(* CODESYS project cylinders_initial.project

Project tree, tasks and I/O mapping:
  Device : CODESYS Control Win V3, 3S - Smart Software Solutions GmbH, version 3.5.16.0
    application Application
      libraries: Standard, * (System); CmpBitmapPool, * (System); Util, * (System)
      task MainTask (cyclic, interval 5 ms, priority 1) calls cylinder_ctrl_SFC
      task simulation (cyclic, interval t#20ms, priority 1) calls sim_logic
      task VISU_TASK (cyclic, interval 10 ms, priority 31) calls VisuElems.Visu_Prg
      visualisation Cylinders
      global variables IO
      control/
        program cylinder_ctrl [LD]
        function block CylinderFB [LD]
        function block LampCTRL [SFC]
        program cylinder_ctrl_SFC [LD]
        function block Sequence [SFC]
      simulation/
        program sim_logic [LD]
        function block cylSimulation [ST]
      image pool ImagePool
  libraries: VisuSymbols, 3.5.10.0 (System)
  5ce3da45-db07-42e7-a21c-a00fff4ed8f6|C:\Users\ryytt\OneDrive\Skrivbord\examensarbete\bakgrund.png
  5ce3da45-db07-42e7-a21c-a00fff4ed8f6|C:\Users\ryytt\OneDrive\Skrivbord\examensarbete\bakgrundv2.png
  text list GlobalTextList
*)

// Device/Application/IO
VAR_GLOBAL
	ixStart: BOOL; // the start switch and the button
 	ixStop: BOOL;  // the stop switch and the button
	ixReset: BOOL; // the reset switch
	ixB1: BOOL; // button B1
	ixB2: BOOL; // button B2
	ixIN10: BOOL; // the IN10 switch
	ixIN11: BOOL; // the IN11 switch
	ixCylinder1In: BOOL; // a sensor if cylinder 1 is in
	ixCylinder1Out: BOOL; // a sensor if cylinder 1 is in
	ixCylinder2In: BOOL; // a sensor if cylinder 1 is in
	ixCylinder2Out: BOOL; // a sensor if cylinder 1 is in
	ixCylinder3In: BOOL; // a sensor if cylinder 1 is in
	ixCylinder3Out: BOOL; // a sensor if cylinder 1 is in	
	ixEmergencyStop: BOOL := TRUE; // the emergency stop. If false, it is active

	qxLamp1: BOOL; // to control L1
	qxLamp2: BOOL; // to control L2
	qxLamp3: BOOL; // to ontorl L3
	qxLamp4: BOOL; // to control L4
	qxCylinder1: BOOL; // to extend cylinder 1
	qxCylinder2: BOOL; // to extend cylinder 2
	qxCylinder3: BOOL; // to extend cylinder 3
	ixCylinderIn_cyl23: BOOL;
	ixCylinderOut_cyl23: BOOL;
END_VAR

// Device/Application/control/cylinder_ctrl_SFC
PROGRAM cylinder_ctrl_SFC
VAR
	cylinder1: CylinderFB;
	cylinder2: CylinderFB;
	cylinder3: CylinderFB;
	
	sequence_ctrl1: Sequence;
	sequence_ctrl23: Sequence;
	
	LampCTRL_0: LampCTRL;
	lamp_testing: LampCTRL;
END_VAR

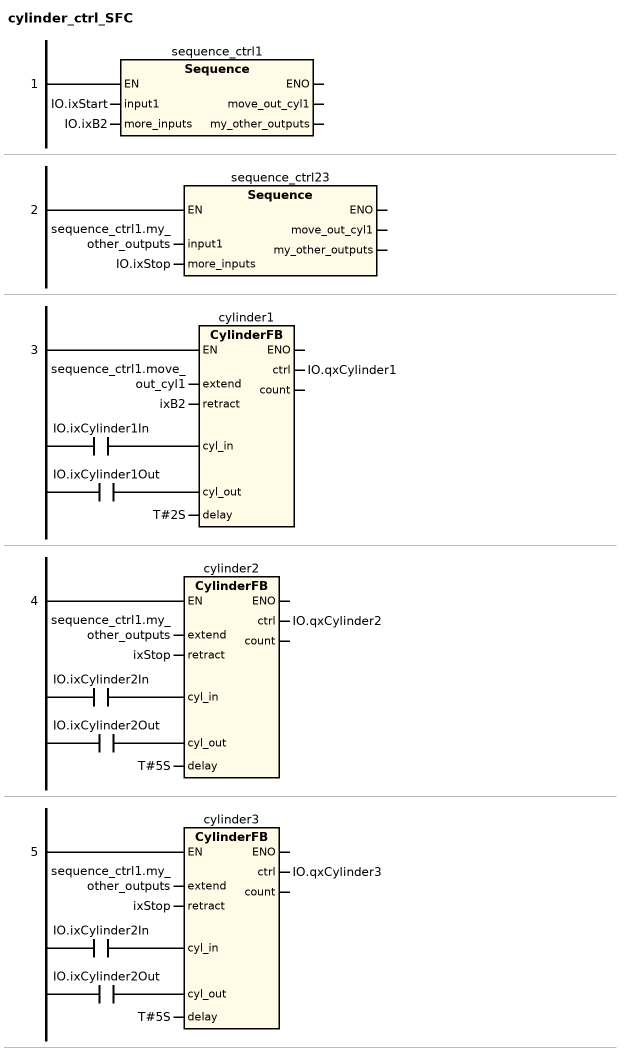
// NETWORK 1
sequence_ctrl1(input1 := IO.ixStart, more_inputs := IO.ixB2); // Sequence

// NETWORK 2
sequence_ctrl23(input1 := sequence_ctrl1.my_other_outputs, more_inputs := IO.ixStop); // Sequence

// NETWORK 3
cylinder1(
    extend := sequence_ctrl1.move_out_cyl1,
    retract := ixB2,
    cyl_in := IO.ixCylinder1In,
    cyl_out := IO.ixCylinder1Out,
    delay := T#2S,
    ctrl => IO.qxCylinder1); // CylinderFB

// NETWORK 4
cylinder2(
    extend := sequence_ctrl1.my_other_outputs,
    retract := ixStop,
    cyl_in := IO.ixCylinder2In,
    cyl_out := IO.ixCylinder2Out,
    delay := T#5S,
    ctrl => IO.qxCylinder2); // CylinderFB

// NETWORK 5
cylinder3(
    extend := sequence_ctrl1.my_other_outputs,
    retract := ixStop,
    cyl_in := IO.ixCylinder2In,
    cyl_out := IO.ixCylinder2Out,
    delay := T#5S,
    ctrl => IO.qxCylinder3); // CylinderFB

END_PROGRAM

// Device/Application/control/Sequence
FUNCTION_BLOCK Sequence
VAR_INPUT
	input1: BOOL;
	more_inputs: BOOL;
END_VAR
VAR_OUTPUT
	move_out_cyl1: BOOL;
	my_other_outputs: BOOL;
END_VAR
VAR
	init: BOOL := TRUE;
END_VAR

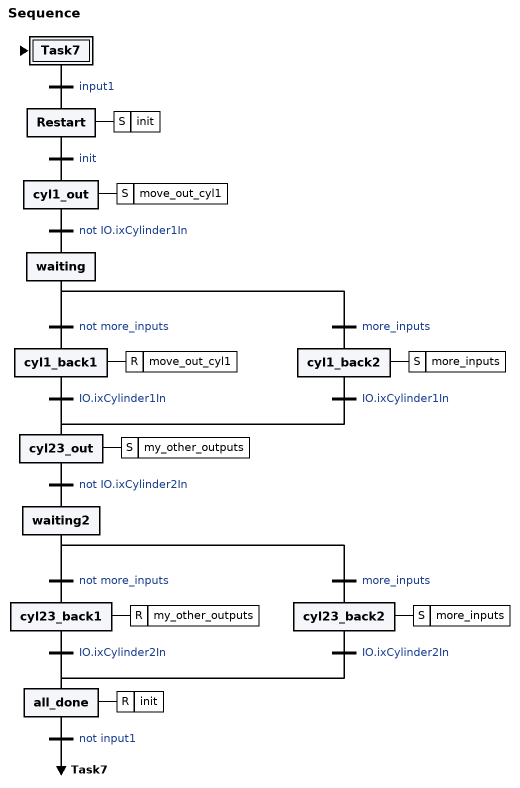
INITIAL_STEP Task7:
END_STEP
TRANSITION FROM Task7 TO Restart
    := input1;
END_TRANSITION
STEP Restart:
    init(S);
END_STEP
TRANSITION FROM Restart TO cyl1_out
    := init;
END_TRANSITION
STEP cyl1_out:
    move_out_cyl1(S);
END_STEP
TRANSITION FROM cyl1_out TO waiting
    := not IO.ixCylinder1In;
END_TRANSITION
STEP waiting:
END_STEP
TRANSITION FROM waiting TO cyl1_back1
    := not more_inputs;
END_TRANSITION
STEP cyl1_back1:
    move_out_cyl1(R);
END_STEP
TRANSITION FROM cyl1_back1 TO cyl23_out
    := IO.ixCylinder1In;
END_TRANSITION
TRANSITION FROM waiting TO cyl1_back2
    := more_inputs;
END_TRANSITION
STEP cyl1_back2:
    more_inputs(S);
END_STEP
TRANSITION FROM cyl1_back2 TO cyl23_out
    := IO.ixCylinder1In;
END_TRANSITION
STEP cyl23_out:
    my_other_outputs(S);
END_STEP
TRANSITION FROM cyl23_out TO waiting2
    := not IO.ixCylinder2In;
END_TRANSITION
STEP waiting2:
END_STEP
TRANSITION FROM waiting2 TO cyl23_back1
    := not more_inputs;
END_TRANSITION
STEP cyl23_back1:
    my_other_outputs(R);
END_STEP
TRANSITION FROM cyl23_back1 TO all_done
    := IO.ixCylinder2In;
END_TRANSITION
TRANSITION FROM waiting2 TO cyl23_back2
    := more_inputs;
END_TRANSITION
STEP cyl23_back2:
    more_inputs(S);
END_STEP
TRANSITION FROM cyl23_back2 TO all_done
    := IO.ixCylinder2In;
END_TRANSITION
STEP all_done:
    init(R);
END_STEP
TRANSITION FROM all_done TO Task7
    := not input1;
END_TRANSITION

END_FUNCTION_BLOCK

// Device/Application/control/CylinderFB
FUNCTION_BLOCK CylinderFB
VAR_INPUT
	extend: BOOL;	// signal to extend. Extends on positive edge
	retract: BOOL;	// signal to retract
	cyl_in: BOOL;	// sensor that cylinder is not extended, i.e. in
	cyl_out: BOOL;	// sensor that cylinder is not extended, i.e. in
	delay: TIME;
END_VAR
VAR_OUTPUT
	ctrl: BOOL;	// sensor that cylinder is not extended, i.e. in
	count: INT :=0;	// times the cylinder has been extended (cyl_out became true)
END_VAR
VAR
	ton_cyl1: TON;

	ton_cyl23: TON;
	stop: BOOL;
	converstion: BOOL;
	
	t: INT :=5;
END_VAR
VAR // added by the converter: edge detectors and wires of the graphical bodies
    _rt1 : R_TRIG;
END_VAR

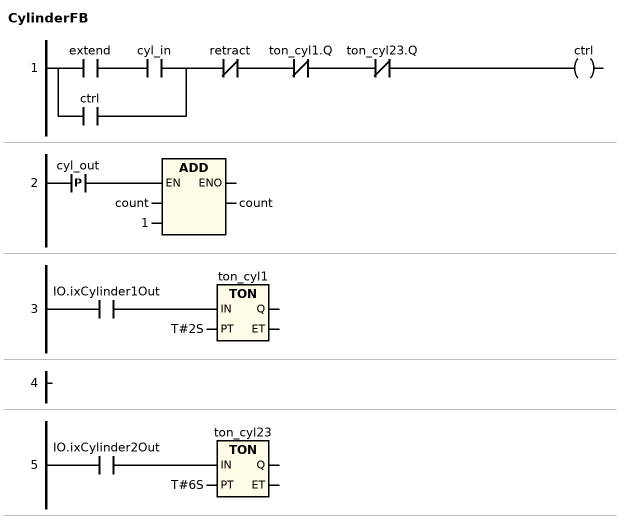
// NETWORK 1
ctrl := (extend AND cyl_in OR ctrl) AND NOT retract AND NOT ton_cyl1.Q AND NOT ton_cyl23.Q;

// NETWORK 2
_rt1(CLK := cyl_out);
IF _rt1.Q THEN count := count + 1; END_IF

// NETWORK 3
ton_cyl1(IN := IO.ixCylinder1Out, PT := T#2S); // TON

// NETWORK 4

// NETWORK 5
ton_cyl23(IN := IO.ixCylinder2Out, PT := T#6S); // TON

END_FUNCTION_BLOCK

// Device/Application/control/LampCTRL
FUNCTION_BLOCK LampCTRL
VAR_INPUT
	start: BOOL;
END_VAR
VAR_OUTPUT
	l1: BOOL;
	l2: BOOL;
	l3: BOOL;
	l4: BOOL;
END_VAR
VAR
END_VAR

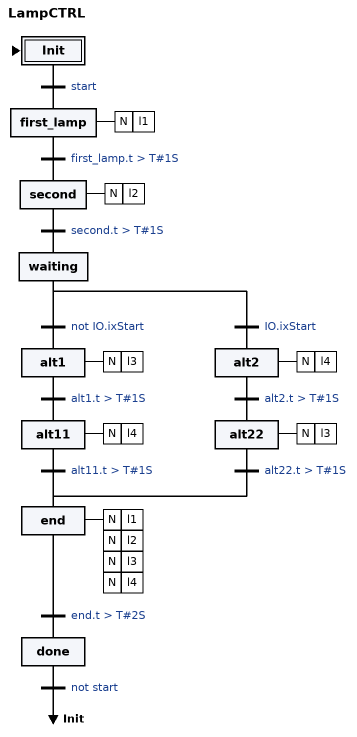
INITIAL_STEP Init:
END_STEP
TRANSITION FROM Init TO first_lamp
    := start;
END_TRANSITION
STEP first_lamp:
    l1(N);
END_STEP
TRANSITION FROM first_lamp TO second
    := first_lamp.t > T#1S;
END_TRANSITION
STEP second:
    l2(N);
END_STEP
TRANSITION FROM second TO waiting
    := second.t > T#1S;
END_TRANSITION
STEP waiting:
END_STEP
TRANSITION FROM waiting TO alt1
    := not IO.ixStart;
END_TRANSITION
STEP alt1:
    l3(N);
END_STEP
TRANSITION FROM alt1 TO alt11
    := alt1.t > T#1S;
END_TRANSITION
STEP alt11:
    l4(N);
END_STEP
TRANSITION FROM alt11 TO end
    := alt11.t > T#1S;
END_TRANSITION
TRANSITION FROM waiting TO alt2
    := IO.ixStart;
END_TRANSITION
STEP alt2:
    l4(N);
END_STEP
TRANSITION FROM alt2 TO alt22
    := alt2.t > T#1S;
END_TRANSITION
STEP alt22:
    l3(N);
END_STEP
TRANSITION FROM alt22 TO end
    := alt22.t > T#1S;
END_TRANSITION
STEP end:
    l1(N);
    l2(N);
    l3(N);
    l4(N);
END_STEP
TRANSITION FROM end TO done
    := end.t > T#2S;
END_TRANSITION
STEP done:
END_STEP
TRANSITION FROM done TO Init
    := not start;
END_TRANSITION

END_FUNCTION_BLOCK

// Device/Application/simulation/sim_logic
PROGRAM sim_logic
VAR
	cyl1: cylSimulation;
	donotuse_cyl1_pos: INT;
	cyl2: cylSimulation;
	cyl3: cylSimulation;
	donotuse_cyl2_pos: INT;
	donotuse_cyl3_pos: INT;
END_VAR

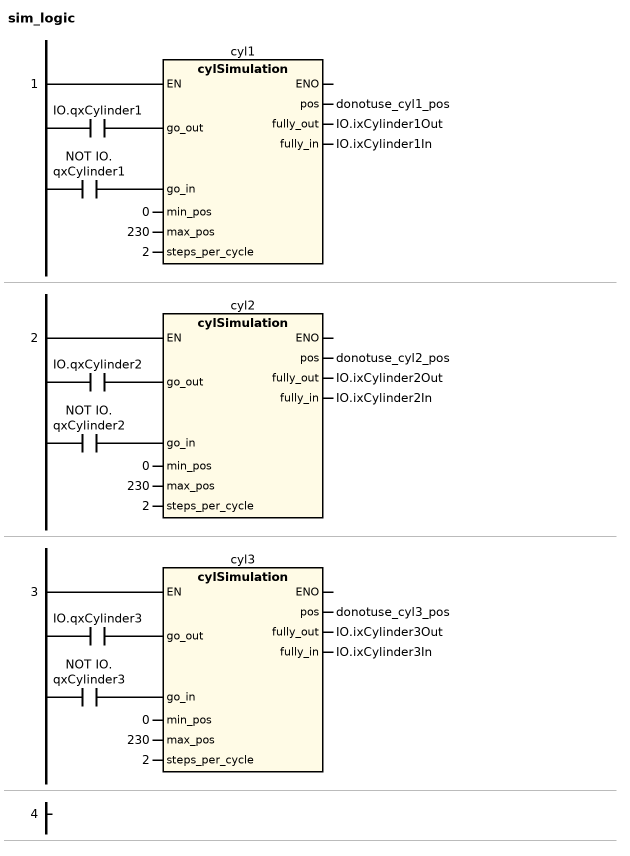
// NETWORK 1
cyl1(
    go_out := IO.qxCylinder1,
    go_in := NOT IO.qxCylinder1,
    min_pos := 0,
    max_pos := 230,
    steps_per_cycle := 2,
    pos => donotuse_cyl1_pos,
    fully_out => IO.ixCylinder1Out,
    fully_in => IO.ixCylinder1In); // cylSimulation

// NETWORK 2
cyl2(
    go_out := IO.qxCylinder2,
    go_in := NOT IO.qxCylinder2,
    min_pos := 0,
    max_pos := 230,
    steps_per_cycle := 2,
    pos => donotuse_cyl2_pos,
    fully_out => IO.ixCylinder2Out,
    fully_in => IO.ixCylinder2In); // cylSimulation

// NETWORK 3
cyl3(
    go_out := IO.qxCylinder3,
    go_in := NOT IO.qxCylinder3,
    min_pos := 0,
    max_pos := 230,
    steps_per_cycle := 2,
    pos => donotuse_cyl3_pos,
    fully_out => IO.ixCylinder3Out,
    fully_in => IO.ixCylinder3In); // cylSimulation

// NETWORK 4

END_PROGRAM

// Device/Application/simulation/cylSimulation
FUNCTION_BLOCK cylSimulation
VAR_INPUT
	go_out: BOOL;
	go_in: BOOL;
	min_pos: INT;
	max_pos: INT;
	steps_per_cycle: INT;
END_VAR
VAR_OUTPUT
	pos: INT;
	fully_out: BOOL;
	fully_in: BOOL;
END_VAR
VAR
END_VAR


IF go_out AND NOT go_in THEN
	pos := pos + steps_per_cycle;
END_IF
IF go_in AND NOT go_out THEN
	pos := pos - steps_per_cycle;
END_IF

pos := LIMIT(min_pos, pos, max_pos);

fully_in := pos = min_pos;
fully_out := pos = max_pos;

END_FUNCTION_BLOCK

// Device/Application/control/cylinder_ctrl
PROGRAM cylinder_ctrl
VAR
	cylinder1: CylinderFB;
	cylinder2: CylinderFB;
	cylinder3: CylinderFB;
	
	init: BOOL := TRUE;
	starting: BOOL;
	cy1_1_out: BOOL;
	cy1_1_done: BOOL;
	
	starting23: BOOL;
	cy1_23_out: BOOL;
	cy1_23_done: BOOL;
		
	LampCTRL_0: LampCTRL;
	lamp_testing: LampCTRL;
END_VAR
VAR // added by the converter: edge detectors and wires of the graphical bodies
    _rt1 : R_TRIG;
    _w1, _w2, _w3, _w4, _w5 : BOOL;
    _ft1 : F_TRIG;
END_VAR

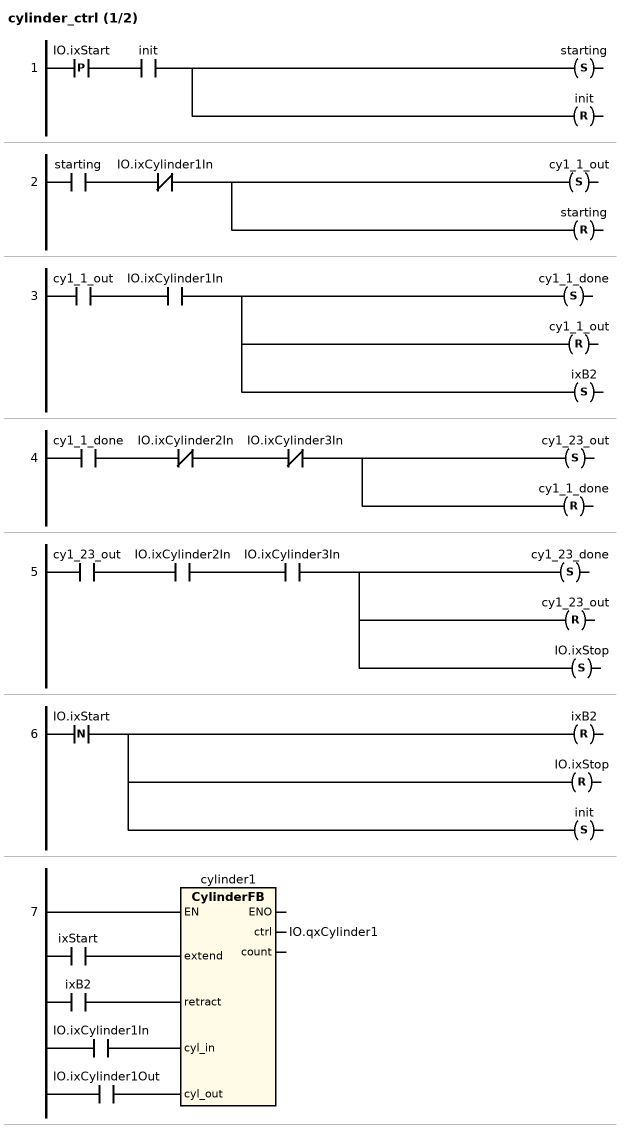
// NETWORK 1
_rt1(CLK := IO.ixStart);
_w1 := _rt1.Q AND init;
starting S= _w1;
init R= _w1;

// NETWORK 2
_w2 := starting AND NOT IO.ixCylinder1In;
cy1_1_out S= _w2;
starting R= _w2;

// NETWORK 3
_w3 := cy1_1_out AND IO.ixCylinder1In;
cy1_1_done S= _w3;
cy1_1_out R= _w3;
ixB2 S= _w3;

// NETWORK 4
_w4 := cy1_1_done AND NOT IO.ixCylinder2In AND NOT IO.ixCylinder3In;
cy1_23_out S= _w4;
cy1_1_done R= _w4;

// NETWORK 5
_w5 := cy1_23_out AND IO.ixCylinder2In AND IO.ixCylinder3In;
cy1_23_done S= _w5;
cy1_23_out R= _w5;
IO.ixStop S= _w5;

// NETWORK 6
_ft1(CLK := IO.ixStart);
ixB2 R= _ft1.Q;
IO.ixStop R= _ft1.Q;
init S= _ft1.Q;

// NETWORK 7
cylinder1(
    extend := ixStart,
    retract := ixB2,
    cyl_in := IO.ixCylinder1In,
    cyl_out := IO.ixCylinder1Out,
    ctrl => IO.qxCylinder1); // CylinderFB

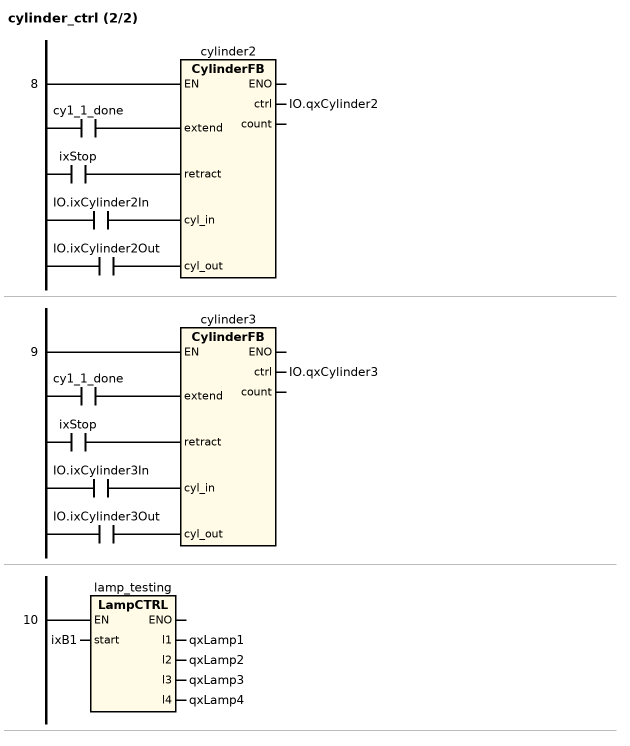
// NETWORK 8
cylinder2(
    extend := cy1_1_done,
    retract := ixStop,
    cyl_in := IO.ixCylinder2In,
    cyl_out := IO.ixCylinder2Out,
    ctrl => IO.qxCylinder2); // CylinderFB

// NETWORK 9
cylinder3(
    extend := cy1_1_done,
    retract := ixStop,
    cyl_in := IO.ixCylinder3In,
    cyl_out := IO.ixCylinder3Out,
    ctrl => IO.qxCylinder3); // CylinderFB

// NETWORK 10
lamp_testing(start := ixB1, l1 => qxLamp1, l2 => qxLamp2, l3 => qxLamp3, l4 => qxLamp4); // LampCTRL

END_PROGRAM

// Device/Application/Cylinders
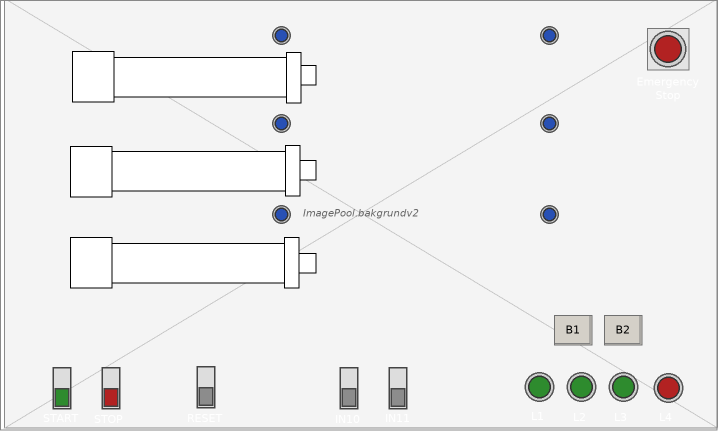
VISUALIZATION Cylinders  // 718x431
    Image (4,-2 714x430), image: ImagePool.bakgrundv2
    Rectangle (286,253 30x20)
        p874137650: sim_logic.donotuse_cyl3_pos
    Rectangle (286,160 30x20)
        p874137650: sim_logic.donotuse_cyl2_pos
    Lamp1 (522,370 35x34), tooltip "L1", variable: qxLamp1, style: Lamp-Lamp1-Green
    Lamp1 (564,370 35x34), tooltip "L2", variable: qxLamp2, style: Lamp-Lamp1-Green
    Lamp1 (606,370 35x34), tooltip "L3", variable: qxLamp3, style: Lamp-Lamp1-Green
    Lamp1 (651,371 35x34), tooltip "L4", variable: qxLamp4, style: Lamp-Lamp1-Red
    DipSwitch (41,366 42x44), variable: ixStart, behaviour: TOGGLE, style: Switch-DipSwitch-Green
    DipSwitch (90,366 42x44), variable: ixStop, behaviour: TOGGLE, style: Switch-DipSwitch-Red
    DipSwitch (185,365 42x44), tooltip "RESET", variable: ixReset, behaviour: TOGGLE, style: Switch-DipSwitch-Gray
    DipSwitch (328,366 42x44), variable: ixIN10, behaviour: TOGGLE, style: Switch-DipSwitch-Gray
    DipSwitch (377,366 42x44), variable: ixIN11, behaviour: TOGGLE, style: Switch-DipSwitch-Gray
    Label (16,409 89x19), "START"
    Label (64,410 89x19), "STOP"
    Label (160,409 89x19), "RESET"
    Label (303,410 89x19), "IN10"
    Label (353,409 89x19), "IN11"
    Label (493,407 89x19), "L1"
    Label (535,408 89x19), "L2"
    Label (576,408 89x19), "L3"
    Label (621,408 89x19), "L4"
    Rectangle (286,65 30x20)
        p874137650: sim_logic.donotuse_cyl1_pos
    Rectangle (101,57 193x40)
    Rectangle (99,151 193x40)
    Rectangle (102,243 193x40)
    RoundedRectangle (70,237 42x51), "CYL3"
    RoundedRectangle (70,146 42x51), "CYL2"
    RoundedRectangle (72,51 42x51), "CYL1"
    RoundedRectangle (286,52 15x51)
    RoundedRectangle (285,145 15x51)
    RoundedRectangle (284,237 15x51)
    Lamp1 (271,25 21x21), variable: ixCylinder1In, style: Lamp-Lamp1-Blue
    Lamp1 (539,25 21x21), variable: ixCylinder1Out, style: Lamp-Lamp1-Blue
    Lamp1 (271,113 21x21), variable: ixCylinder2In, style: Lamp-Lamp1-Blue
    Lamp1 (539,113 21x21), variable: ixCylinder2Out, style: Lamp-Lamp1-Blue
    Lamp1 (271,204 21x21), variable: ixCylinder3In, style: Lamp-Lamp1-Blue
    Lamp1 (539,204 21x21), variable: ixCylinder3Out, style: Lamp-Lamp1-Blue
    PushSwitch (647,27 42x44), variable: ixEmergencyStop, behaviour: TOGGLE, style: Switch-PushSwitch-Red
    Label (623,72 90x33), "Emergency Stop"
    Button (554,315 38x30), "B1"
        tap ixB1
    Button (604,315 38x30), "B2"
        tap ixB2
END_VISUALIZATION
